Universal Robots PolyScope program: socket-send-waypoints.urp

Program socket-send-waypoints (createdIn=3.4.5.437 lastSavedIn=3.5.3.10825 directory=/home/ur/ursim-current/programs installation=default robotSerialNumber=2014359999)
Calibrated DH parameters: a=[0.000051, -0.034486, -0.39219, -0.000006, 0.000147, 0]; d=[0.089266, 223.105289, -223.633213, 0.638611, 0.094791, 0.082527]; alpha=[1.569365, -0.0019, 0.014195, 1.569882, -1.569779, 0]; deltaTheta=[0.000016, -1.489587, 1.470486, 0.019132, -0.000025, -0.000047]
Robot Program (runOnlyOnce=true motionType=MoveJ speed=1.047198 acceleration=1.396263 useActiveTCP=false)
  Script: set_tcp(p[0,0,0.067,0,0,0])
  Script: set_standard_digital_out(0,False)
  Script: movej([0.0102974,-1.52506,1.68598,-1.73084,-1.5547,1.58406],a=0.1,v=0.25)
  Script: socket = socket_open("192.168.1.101", 30002, "socket_0")
  If socket (checkContinuously=true)
    Script: socket_send_int(0, "socket_0")
    Script: points = socket_read_ascii_float(1,"socket_0")
    Script: counter = 1
    Loop While (checkContinuously=false) expression=counter ≤ points[1]
      Script: socket_send_int(counter, "socket_0")
      Script: traj = socket_read_ascii_float(7, "socket_0")
      Script: servoj(get_inverse_kin(p[traj[1],traj[2],traj[3],traj[4],traj[5],traj[6]]),t=traj[7])
      Script: counter = counter + 1
    Script: midpoint = get_actual_tcp_pose()
    Script: socket_send_int(999,"socket_0")
    Script: target = socket_read_ascii_float(6,"socket_0")
    Script: movel(p[target[1],target[2],target[3],target[4],target[5],target[6]],a=0.1,v=0.25)
    Script: set_standard_digital_out(0,True)
    Wait Sleep waitTime=0.2
    Script: movel(midpoint,a=0.1,v=0.25)
    Script: movej([0.0102974,-1.52506,1.68598,-1.73084,-1.5547,1.58406],a=0.1,v=0.25)
    Script: socket_send_int(777, "socket_0")
    Wait Sleep waitTime=2
    Script: socket_close("socket_0")
  Else 
    Wait Sleep waitTime=1
